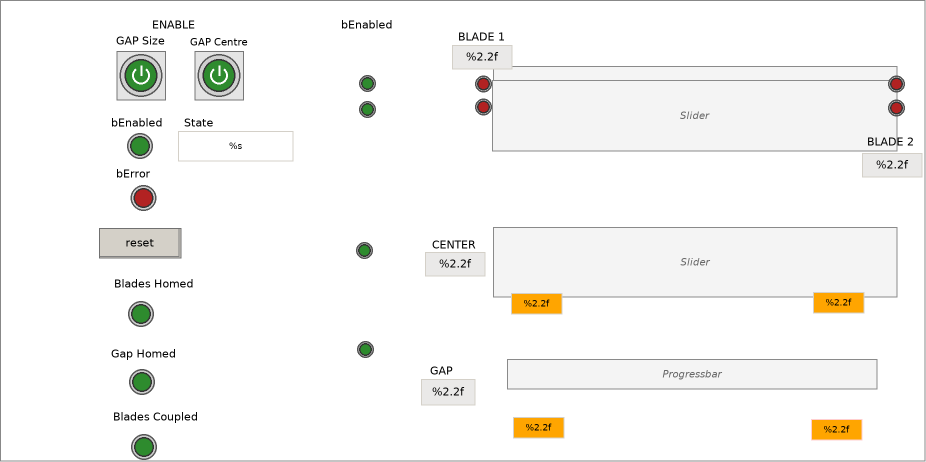
VISUALIZATION SlitsVisuVertical  // 926x462
    Slider (493,66 404x74), variable: astAxes[1].Axis.NcToPlc.ActPos, scale -90..90
    Slider (492,80 405x71), variable: astAxes[2].Axis.NcToPlc.ActPos, scale -90..90
    Slider (493,227 404x70), variable: astAxes[4].Axis.NcToPlc.ActPos, scale -90..90
    Progressbar (507,359 370x30), variable: astAxes[3].Axis.NcToPlc.ActPos
    PowerSwitch (116,51 50x49), variable: GVL.astAxes[ymir_slits.fbSlitVertical.iGapSize].stControl.bEnable, behaviour: TOGGLE, style: Switch-PowerSwitch-Green
    Textfield (149,13 62x24), "ENABLE", text index: "enable"
    Lamp1 (125,131 30x30), variable: ymir_slits.fbSlitVertical.bEnabled, style: Lamp-Lamp1-Green
    Textfield (108,108 60x30), "bEnabled", text list: "languageSupport", text index: "bEnabled"
    Lamp1 (126,299 30x30), variable: ymir_slits.fbSlitVertical.bBladesHomed, style: Lamp-Lamp1-Green
    Lamp1 (129,432 30x30), variable: ymir_slits.fbSlitVertical.bBladesCoupled, style: Lamp-Lamp1-Green
    Textfield (110,402 104x30), "Blades Coupled"
    Textfield (111,269 97x30), "Blades Homed", text list: ''
    Lamp1 (474,73 19x22), variable: GVL.astAxes[1].stInputs.bLimitBwd, style: Lamp-Lamp1-Red
    Lamp1 (474,96 19x22), variable: GVL.astAxes[2].stInputs.bLimitBwd, style: Lamp-Lamp1-Red
    Lamp1 (887,97 19x22), variable: GVL.astAxes[2].stInputs.bLimitFwd, style: Lamp-Lamp1-Red
    Lamp1 (887,73 19x22), variable: GVL.astAxes[1].stInputs.bLimitFwd, style: Lamp-Lamp1-Red
    Lamp1 (125,183 37x30), variable: ymir_slits.fbSlitVertical.eSlitPairState, style: Lamp-Lamp1-Red
    Textfield (113,159 120x30), "bError", text list: "languageSupport", text index: "bError"
    Button (99,228 82x30), "reset", pressed state: ymir_slits.fbSlitVertical.bReset
        OnMouseClick: toggle ymir_slits.fbSlitVertical.bReset
    Textfield (455,25 62x24), "BLADE 1"
    Textfield (864,130 62x24), "BLADE 2", text index: "enable"
    Textfield (429,233 62x24), "CENTER"
    Textfield (427,359 62x24), "GAP", text index: "enable"
    Textfield (178,131 115x30), "%s", text variable: ymir_slits.fbSlitVertical.eSlitPairState
    Textfield (181,108 60x30), "State"
    Textfield (425,252 60x24), "%2.2f", text variable: GVL.astAxes[ymir_slits.fbSlitVertical.iGapCentre].stStatus.fActPosition
    Textfield (421,379 54x26), "%2.2f", text variable: GVL.astAxes[ymir_slits.fbSlitVertical.iGapSize].stStatus.fActPosition
    Lamp1 (358,74 19x19), variable: GVL.astAxes[ymir_slits.fbSlitVertical.iBladeNegative].stStatus.bEnabled, style: Lamp-Lamp1-Green
    Textfield (338,10 60x30), "bEnabled", text list: "languageSupport", text index: "bEnabled"
    Lamp1 (358,100 19x19), variable: GVL.astAxes[ymir_slits.fbSlitVertical.iBladePositive].stStatus.bEnabled, style: Lamp-Lamp1-Green
    Lamp1 (355,241 19x19), variable: GVL.astAxes[ymir_slits.fbSlitVertical.iGapCentre].stStatus.bEnabled, style: Lamp-Lamp1-Green
    Lamp1 (356,340 19x19), variable: GVL.astAxes[ymir_slits.fbSlitVertical.iGapSize].stStatus.bEnabled, style: Lamp-Lamp1-Green
    Lamp1 (127,367 30x30), variable: ymir_slits.fbSlitVertical.bGapHomed, style: Lamp-Lamp1-Green
    Textfield (108,339 97x30), "Gap Homed", text list: ''
    Textfield (511,293 51x21), "%2.2f", text variable: GVL.astAxes[ymir_slits.fbSlitVertical.iGapCentre].stConfig.fMinSoftPosLimit
    Textfield (811,419 51x21), "%2.2f", text variable: GVL.astAxes[ymir_slits.fbSlitVertical.iGapSize].stConfig.fMaxSoftPosLimit
    Textfield (813,292 51x21), "%2.2f", text variable: GVL.astAxes[ymir_slits.fbSlitVertical.iGapCentre].stConfig.fMaxSoftPosLimit
    Textfield (513,417 51x21), "%2.2f", text variable: GVL.astAxes[ymir_slits.fbSlitVertical.iGapSize].stConfig.fMinSoftPosLimit
    PowerSwitch (194,51 50x49), variable: GVL.astAxes[ymir_slits.fbSlitVertical.iGapCentre].stControl.bEnable, behaviour: TOGGLE, style: Switch-PowerSwitch-Green
    Textfield (113,29 62x24), "GAP Size", text index: "enable"
    Textfield (187,30 62x24), "GAP Centre", text index: "enable"
    Textfield (452,45 60x24), "%2.2f", text variable: GVL.astAxes[ymir_slits.fbSlitVertical.iBladeNegative].stStatus.fActPosition
    Textfield (862,153 60x24), "%2.2f", text variable: GVL.astAxes[ymir_slits.fbSlitVertical.iBladePositive].stStatus.fActPosition
END_VISUALIZATION

(* stored: Version 1.1.0.1
   Visu SlitsVisuVertical: Id {df576c84-0c17-466f-9725-4d1bca57cd5e} *)
